SUBAPPLICATION Uebung_006a2 (* 2x SR und T-Flip-Flop mit IE *)
  (* Standard: 61499-2; Description: Copyright (c) 2023 Meisterschulen am Ostbahnhof This program and the accompanying materials are made available under the terms of the Eclipse Public License 2.0 which is available at https://www.eclipse.org/legal/epl-2.0/ SPDX-License-Identifier: EPL-2.0 *)
  (* Version 1.0, 2023-10-23, Franz Höpfinger, Meisterschulen am Ostbahnhof *)
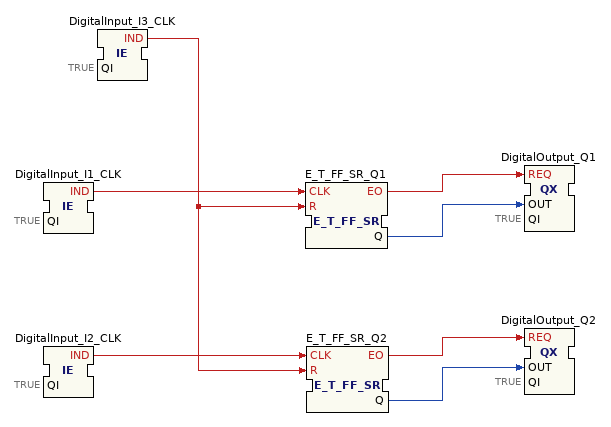
  FBS
    DigitalOutput_Q1 : QX(QI := TRUE);
    DigitalInput_I1_CLK : IE(QI := TRUE);
    DigitalInput_I2_CLK : IE(QI := TRUE);
    E_T_FF_SR_Q1 : E_T_FF_SR;
    DigitalInput_I3_CLK : IE(QI := TRUE);
    E_T_FF_SR_Q2 : E_T_FF_SR;
    DigitalOutput_Q2 : QX(QI := TRUE);
  END_FBS
  EVENT_CONNECTIONS
    E_T_FF_SR_Q1.EO TO DigitalOutput_Q1.REQ;
    E_T_FF_SR_Q2.EO TO DigitalOutput_Q2.REQ;
    DigitalInput_I1_CLK.IND TO E_T_FF_SR_Q1.CLK;
    DigitalInput_I2_CLK.IND TO E_T_FF_SR_Q2.CLK;
    DigitalInput_I3_CLK.IND TO E_T_FF_SR_Q2.R;
    DigitalInput_I3_CLK.IND TO E_T_FF_SR_Q1.R;
  END_CONNECTIONS
  DATA_CONNECTIONS
    E_T_FF_SR_Q1.Q TO DigitalOutput_Q1.OUT;
    E_T_FF_SR_Q2.Q TO DigitalOutput_Q2.OUT;
  END_CONNECTIONS
END_SUBAPPLICATION
